FUNCTION TIME_TO_REAL
  (* Standard: 61499-1 *)
  (* Version 1.0, 2025-12-21, Franz Höpfinger *)
  PACKAGE OSCAT::Basic::POUs::conversion;
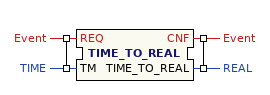
  EVENT_INPUT
    REQ WITH TM;
  END_EVENT
  EVENT_OUTPUT
    CNF WITH TIME_TO_REAL;
  END_EVENT
  VAR_INPUT
    TM : TIME;
  END_VAR
  VAR_OUTPUT
    TIME_TO_REAL : REAL;
  END_VAR
  BODY IN ST:
PACKAGE OSCAT::Basic::POUs::conversion;

FUNCTION TIME_TO_REAL : REAL
VAR_INPUT
	TM : TIME;
END_VAR

TIME_TO_REAL := UDINT_TO_REAL(TIME_IN_MS_TO_UDINT(TM));

END_FUNCTION
  END_BODY
END_FUNCTION
